PROGRAM SYSTEM_RESET
VAR CONSTANT
	TRANSITION_COUNT : INT := 10;
END_VAR

VAR
	cycleCounter : INT;
	state : RESET_STATE;
	
	ERROR_ACKNOWLEDGEMENT_BUTTON_OUT AT %Q* : BOOL;
	ESTOP_RESTART_BUTTON_OUT AT %Q* : BOOL;
END_VAR

IF GV_LIFT.SYSTEM_RESET_BUTTON_IN THEN
	cycleCounter := cycleCounter + 1;
	CASE state OF
		RESET_STATE.IDLE :
			IF(cycleCounter >= TRANSITION_COUNT) THEN
				state := RESET_STATE.ERRACK_ON;
				cycleCounter := 0;
			END_IF
		RESET_STATE.ERRACK_ON :
			ERROR_ACKNOWLEDGEMENT_BUTTON_OUT := TRUE;
			IF(cycleCounter >= TRANSITION_COUNT) THEN
				state := RESET_STATE.ERRACK_OFF;
				cycleCounter := 0;
			END_IF
		RESET_STATE.ERRACK_OFF :
			ERROR_ACKNOWLEDGEMENT_BUTTON_OUT := FALSE;
			IF(cycleCounter >= TRANSITION_COUNT) THEN
				state := RESET_STATE.IDLE2;
				cycleCounter := 0;
			END_IF
		RESET_STATE.IDLE2 :
			IF(cycleCounter >= TRANSITION_COUNT) THEN
				state := RESET_STATE.ESTOP_RESET_ON;
				cycleCounter := 0;
			END_IF
		RESET_STATE.ESTOP_RESET_ON :
			ESTOP_RESTART_BUTTON_OUT := TRUE;
			IF(cycleCounter >= TRANSITION_COUNT) THEN
				state := RESET_STATE.COMPLETE;
				cycleCounter := 0;
			END_IF
		RESET_STATE.COMPLETE :
			ESTOP_RESTART_BUTTON_OUT := FALSE;
	END_CASE
ELSE
	cycleCounter := 0;
	state := RESET_STATE.IDLE;
END_IF

END_PROGRAM

(* stored: Version 1.1.0.1, ProductVersion 3.1.4022.12
   POU SYSTEM_RESET: Id {79ec6cbb-745c-4e4b-894b-dfefb2e21cbe}, SpecialFunc None *)
